{attribute addProperty BoxType "EK1122-0000-0018"}
{attribute addProperty Id "Beckhoff_EK11xxsub_EK1100EK1100_179A0949162A_0001_EK1100_0000_0000EK1100_179A0949162A_0002_EK1100_0000_0001EK1100_179A0949162A_0003_EK1100_0000_0016EK1100_179A0949162A_0004_EK1100_0000_0017EK1100_179A0949162A_0005_EK1100_0000_0018EK1100_179A0949162A_0006_EK1100_0008_0016EK1100_179A0949162A_0009_EK1101_0000_0016EK1101_963BF4D7344.25A_0010_EK1101_0000_0017EK1101_963BF4D7344.25A_0011_EK1101_0000_0018EK1101_963BF4D7344.25A_0012_EK1101_0008_0016EK1101_963BF4D7344.25A_0013_EK1101_0010_0016EK1101_963BF4D7344.25A_0008_EK1100_0030_0017EK1100_179A0949162A_0007_EK1100_0030_0016EK1100_179A0949162"}
{attribute addProperty CRC "261757061"}
{attribute addProperty SizeInBites "314"}
{attribute addProperty SizeInBytes "39.25"}
TYPE Beckhoff_EK11xxEK1122_0F9A1885 EXTENDS EK1122_179A0949 :
STRUCT
	{attribute addProperty Name "Beckhoff_EK11xxsub_EK1100"}
	Beckhoff_EK11xxsub_EK1100 : EK1100_179A0949;
	{attribute addProperty Name "A_0001_EK1100_0000_0000"}
	A_0001_EK1100_0000_0000 : EK1100_179A0949;
	{attribute addProperty Name "A_0002_EK1100_0000_0001"}
	A_0002_EK1100_0000_0001 : EK1100_179A0949;
	{attribute addProperty Name "A_0003_EK1100_0000_0016"}
	A_0003_EK1100_0000_0016 : EK1100_179A0949;
	{attribute addProperty Name "A_0004_EK1100_0000_0017"}
	A_0004_EK1100_0000_0017 : EK1100_179A0949;
	{attribute addProperty Name "A_0005_EK1100_0000_0018"}
	A_0005_EK1100_0000_0018 : EK1100_179A0949;
	{attribute addProperty Name "A_0006_EK1100_0008_0016"}
	A_0006_EK1100_0008_0016 : EK1100_179A0949;
	{attribute addProperty Name "A_0009_EK1101_0000_0016"}
	A_0009_EK1101_0000_0016 : EK1101_963BF4D7;
	{attribute addProperty Name "A_0010_EK1101_0000_0017"}
	A_0010_EK1101_0000_0017 : EK1101_963BF4D7;
	{attribute addProperty Name "A_0011_EK1101_0000_0018"}
	A_0011_EK1101_0000_0018 : EK1101_963BF4D7;
	{attribute addProperty Name "A_0012_EK1101_0008_0016"}
	A_0012_EK1101_0008_0016 : EK1101_963BF4D7;
	{attribute addProperty Name "A_0013_EK1101_0010_0016"}
	A_0013_EK1101_0010_0016 : EK1101_963BF4D7;
	{attribute addProperty Name "A_0008_EK1100_0030_0017"}
	A_0008_EK1100_0030_0017 : EK1100_179A0949;
	{attribute addProperty Name "A_0007_EK1100_0030_0016"}
	A_0007_EK1100_0030_0016 : EK1100_179A0949;
END_STRUCT
END_TYPE

(* stored: Version 1.2.0.0, ProductVersion 3.1.4024.9
   DUT Beckhoff_EK11xxEK1122_0F9A1885: Id {acd53629-dc8f-494f-a663-d5cf23c816d1} *)
